TYPE eTcoRoboticsDistance : 
(
    X := 1,
    Y := 2,
    Z := 3,
    XY := 4,
    XZ := 5,
    YZ := 6,
    XYZ := 7
);
END_TYPE

(* stored: Version 1.1.0.1, ProductVersion 3.1.4024.12
   DUT eTcoRoboticsDistance: Id {9cf2ad50-7802-4051-83af-ab7ede919a5f} *)
